// Mitsubishi GX Works2 project: PLC_GROUP_03   PLC: FX3G

// global labels: Global1
VAR_GLOBAL
  petelOriginal AT D1160 : REAL;
  petelCurrent AT D1100 : REAL;
  lemonOriginal AT D1165 : REAL;
  lemonCurrent AT D1105 : REAL;
  meyatzevOriginal AT D1170 : REAL;
  meyatzevCurrent AT D1110 : REAL;
  dubonimOriginal AT D1175 : REAL;
  dubonimCurrent AT D1115 : REAL;
  light7 AT Y007 : BOOL;
  invalidSample AT M4 : BOOL;
  switch5 AT X005 : BOOL;
  no_mlay AT M0 : BOOL;
  switch7 AT X007 : BOOL;
  start_cycle AT X001 : BOOL;
  start_making AT M20 : BOOL;
  TS_0 AT TS0 : BOOL;
  TC_0 AT TC0 : BOOL;
END_VAR
VAR_GLOBAL CONSTANT
  const_50 : INT := 50;
END_VAR
VAR_GLOBAL
  light0 AT Y000 : BOOL;
  sampling AT D1180 : REAL;
  analog_input AT D8280 : INT;
END_VAR
VAR_GLOBAL CONSTANT
  const_400 : REAL := 400.0;
END_VAR
VAR_GLOBAL
  regular_pack AT M1 : BOOL;
  pinuk_pack AT M2 : BOOL;
  mlay_petel_nidrash AT D1120 : REAL;
  mlay_lemon_nidrash AT D1125 : REAL;
  mlay_meyatzev_nidrash AT D1130 : REAL;
  mlay_dubonim_nidrash AT D1135 : REAL;
  no_mlay_petel AT M10 : BOOL;
  no_mlay_lemon AT M11 : BOOL;
  no_mlay_meyatzev AT M12 : BOOL;
  no_mlay_dubonim AT M13 : BOOL;
  switch2 AT X002 : BOOL;
  cooling AT M22 : BOOL;
  light2 AT Y002 : BOOL;
  TC_1 AT TC1 : BOOL;
  TS_1 AT TS1 : BOOL;
  temp_sensor AT X003 : BOOL;
  cool_petel AT D1140 : REAL;
  cool_lemon AT D1145 : REAL;
  mixing AT M24 : BOOL;
  mix_container AT D1150 : REAL;
  mix_time AT D1210 : REAL;
  TC_4 AT TC4 : BOOL;
  TS_4 AT TS4 : BOOL;
  flashing_indicator AT M30 : BOOL;
  TC_2 AT TC2 : BOOL;
  TS_2 AT TS2 : BOOL;
  flash_1 AT Y005 : BOOL;
  flash_2 AT Y006 : BOOL;
  TC_3 AT TC3 : BOOL;
  TS_3 AT TS3 : BOOL;
  finish_mixing AT M40 : BOOL;
  end_work_day AT M5 : BOOL;
  analog_output AT D8282 : INT;
  stock AT D1155 : REAL;
  stock_num AT D1155 : REAL;
END_VAR

// task Task_01 (event TRUE, interval 0, priority 31): POU_01

PROGRAM POU_01
(* structured ladder/FBD written out as ST: instructions are called as NAME(EN, inputs, outputs); _pN, _eN, _tN stand for wires *)
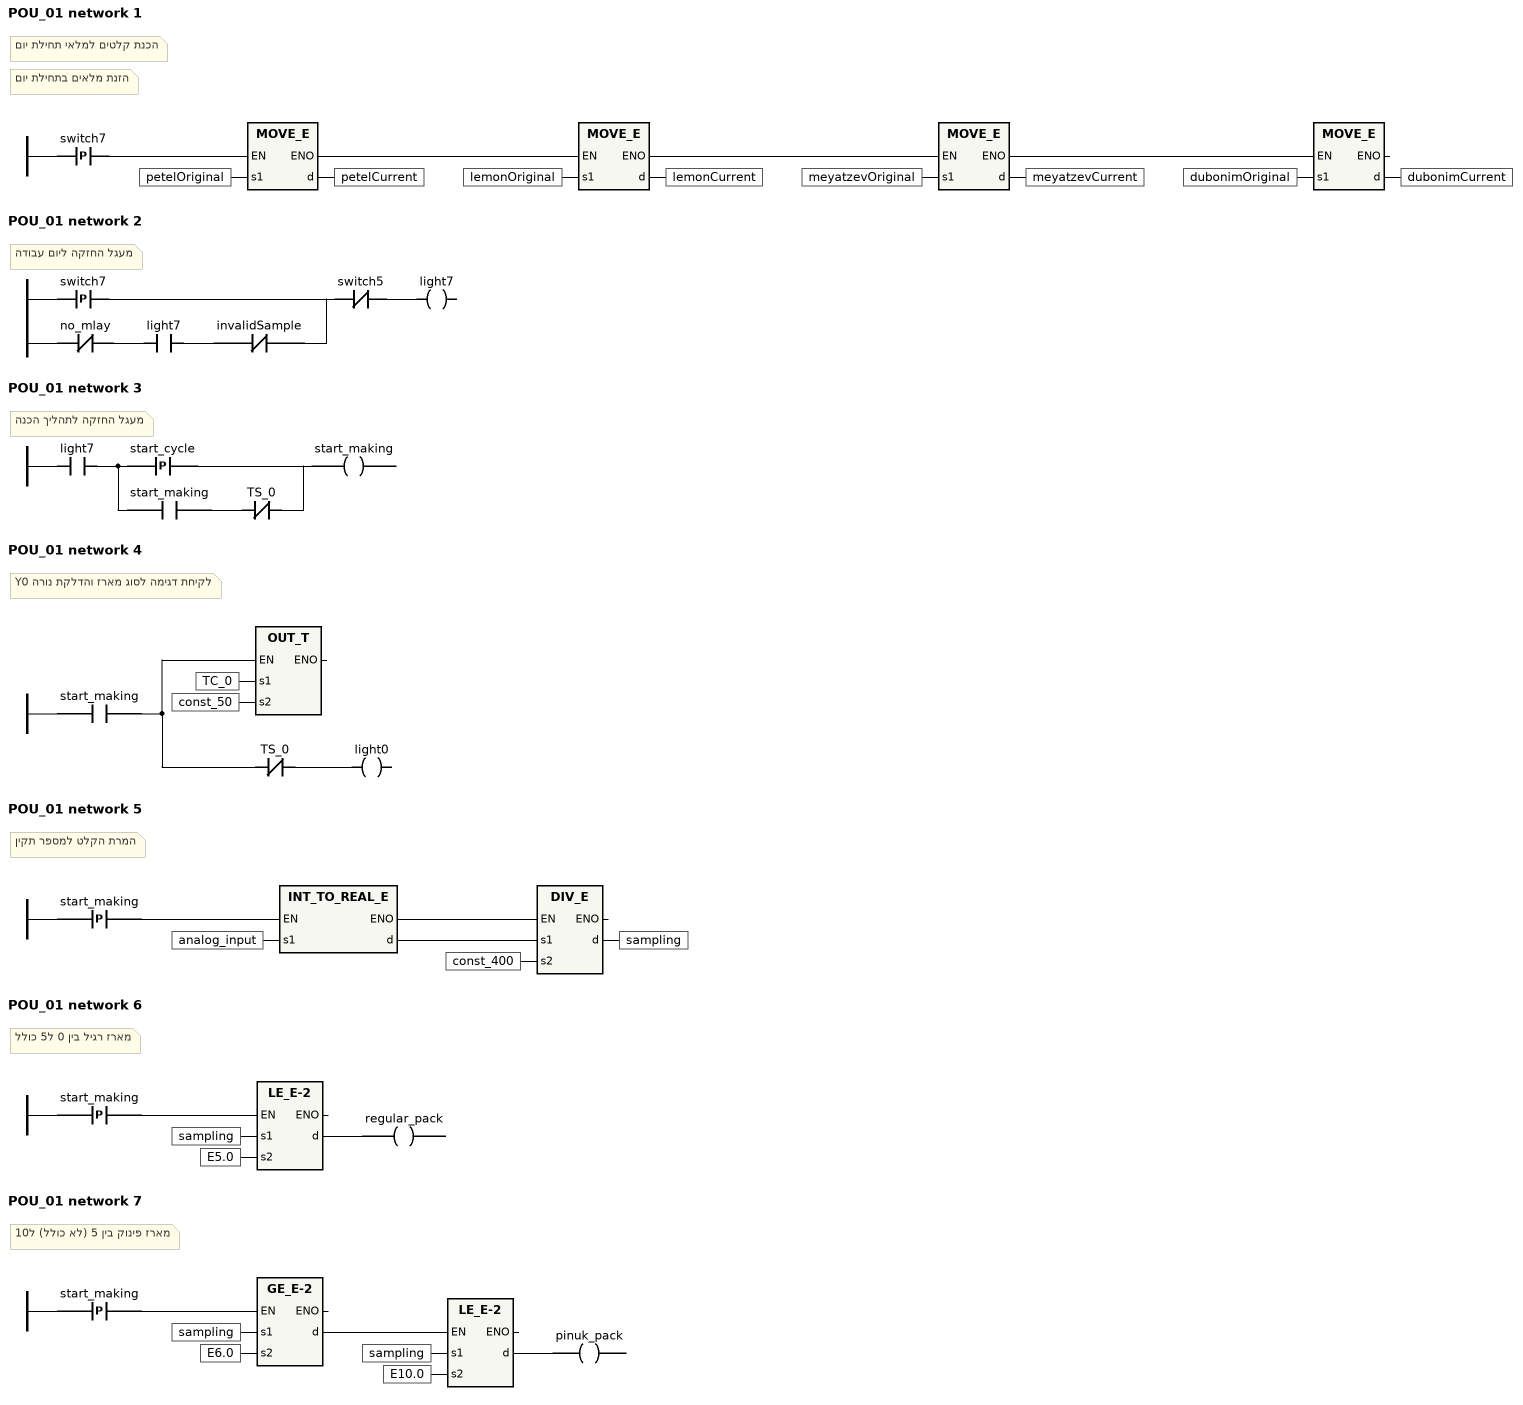
(* network 1 *)
(* הכנת קלטים למלאי תחילת יום *)
(* הזנת מלאים בתחילת יום *)
_e1 := MOVE_E(LDP(TRUE, switch7), petelOriginal, petelCurrent);
_e2 := MOVE_E(_e1, lemonOriginal, lemonCurrent);
_e3 := MOVE_E(_e2, meyatzevOriginal, meyatzevCurrent);
MOVE_E(_e3, dubonimOriginal, dubonimCurrent);
(* network 2 *)
(* מעגל החזקה ליום עבודה *)
light7 := (LDP(TRUE, switch7) OR (NOT no_mlay AND light7 AND NOT invalidSample)) AND NOT switch5;
(* network 3 *)
(* מעגל החזקה לתהליך הכנה *)
start_making := (light7 AND LDP(TRUE, start_cycle)) OR (light7 AND start_making AND NOT TS_0);
(* network 4 *)
(* לקיחת דגימה לסוג מארז והדלקת נורה Y0 *)
OUT_T(start_making, TC_0, const_50);
light0 := start_making AND NOT TS_0;
(* network 5 *)
(* המרת הקלט למספר תקין *)
_e2 := INT_TO_REAL_E(LDP(TRUE, start_making), analog_input, _t1);
DIV_E(_e2, _t1, const_400, sampling);
(* network 6 *)
(* מארז רגיל בין 0 ל5 כולל *)
LE_E(LDP(TRUE, start_making), sampling, E5.0, _t1);
regular_pack := _t1;
(* network 7 *)
(* מארז פינוק בין 5 (לא כולל) ל10 *)
GE_E(LDP(TRUE, start_making), sampling, E6.0, _t1);
LE_E(_t1, sampling, E10.0, _t2);
pinuk_pack := _t2;
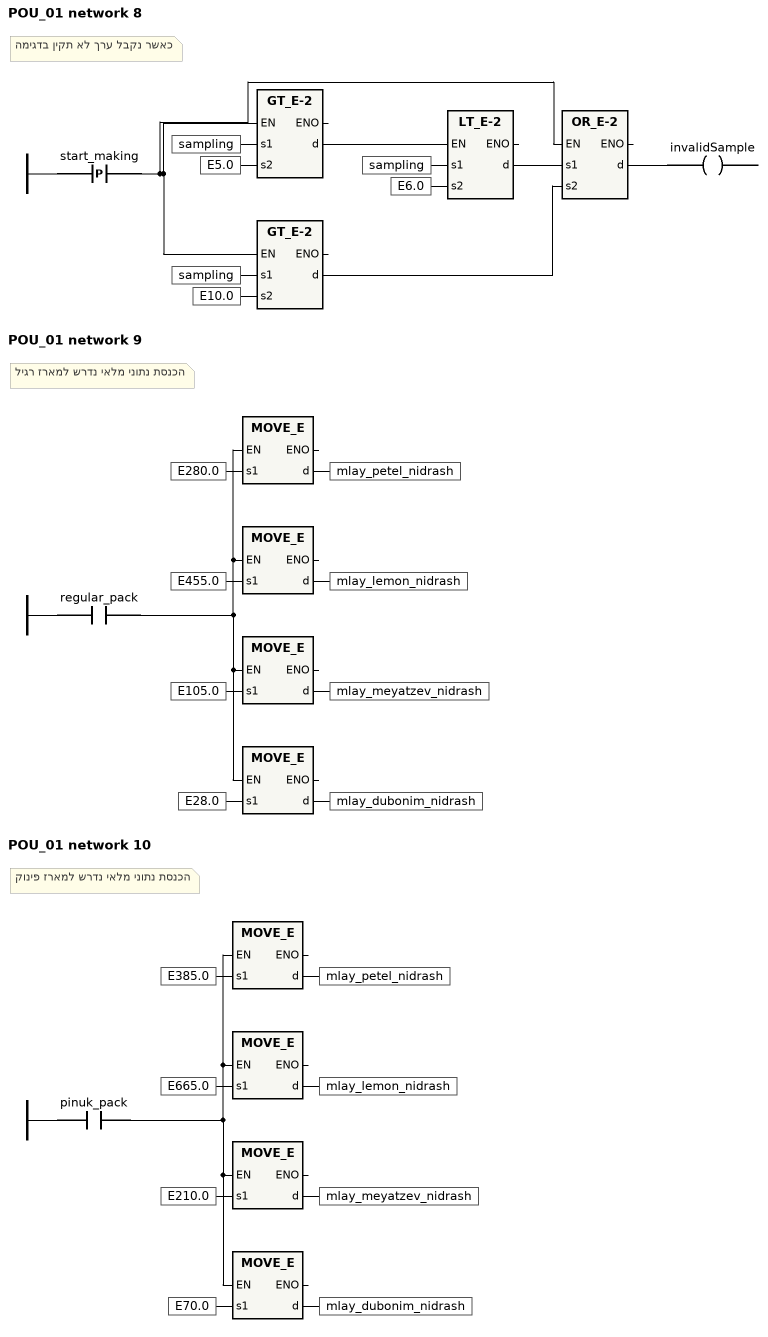
(* network 8 *)
(* כאשר נקבל ערך לא תקין בדגימה *)
_p1 := LDP(TRUE, start_making);
GT_E(_p1, sampling, E5.0, _t2);
LT_E(_t2, sampling, E6.0, _t3);
GT_E(_p1, sampling, E10.0, _t4);
OR_E(_p1, _t3, _t4, _t5);
invalidSample := _t5;
(* network 9 *)
(* הכנסת נתוני מלאי נדרש למארז רגיל *)
MOVE_E(regular_pack, E280.0, mlay_petel_nidrash);
MOVE_E(regular_pack, E455.0, mlay_lemon_nidrash);
MOVE_E(regular_pack, E105.0, mlay_meyatzev_nidrash);
MOVE_E(regular_pack, E28.0, mlay_dubonim_nidrash);
(* network 10 *)
(* הכנסת נתוני מלאי נדרש למארז פינוק *)
MOVE_E(pinuk_pack, E385.0, mlay_petel_nidrash);
MOVE_E(pinuk_pack, E665.0, mlay_lemon_nidrash);
MOVE_E(pinuk_pack, E210.0, mlay_meyatzev_nidrash);
MOVE_E(pinuk_pack, E70.0, mlay_dubonim_nidrash);
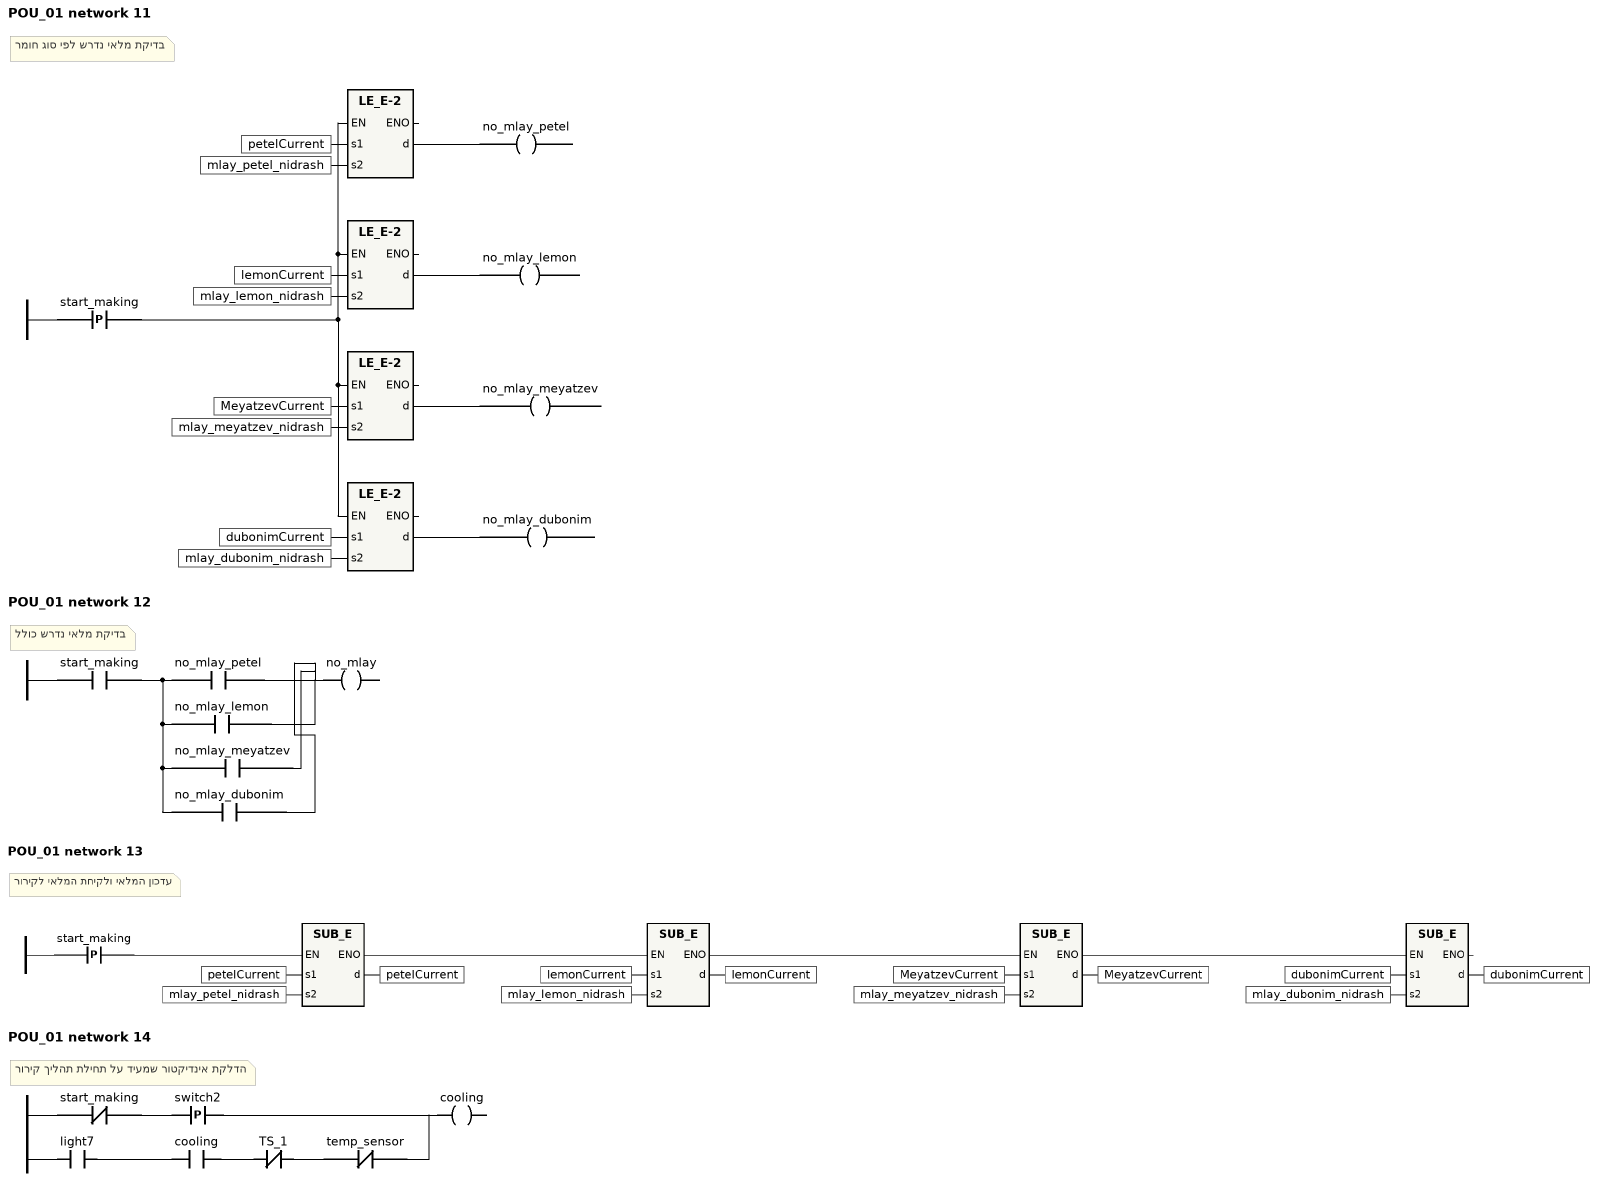
(* network 11 *)
(* בדיקת מלאי נדרש לפי סוג חומר *)
_p1 := LDP(TRUE, start_making);
LE_E(_p1, petelCurrent, mlay_petel_nidrash, _t2);
no_mlay_petel := _t2;
LE_E(_p1, lemonCurrent, mlay_lemon_nidrash, _t3);
no_mlay_lemon := _t3;
LE_E(_p1, MeyatzevCurrent, mlay_meyatzev_nidrash, _t4);
no_mlay_meyatzev := _t4;
LE_E(_p1, dubonimCurrent, mlay_dubonim_nidrash, _t5);
no_mlay_dubonim := _t5;
(* network 12 *)
(* בדיקת מלאי נדרש כולל *)
no_mlay := (start_making AND no_mlay_petel) OR (start_making AND no_mlay_lemon) OR (start_making AND no_mlay_meyatzev) OR (start_making AND no_mlay_dubonim);
(* network 13 *)
(* עדכון המלאי ולקיחת המלאי לקירור *)
_e1 := SUB_E(LDP(TRUE, start_making), petelCurrent, mlay_petel_nidrash, petelCurrent);
_e2 := SUB_E(_e1, lemonCurrent, mlay_lemon_nidrash, lemonCurrent);
_e3 := SUB_E(_e2, MeyatzevCurrent, mlay_meyatzev_nidrash, MeyatzevCurrent);
SUB_E(_e3, dubonimCurrent, mlay_dubonim_nidrash, dubonimCurrent);
(* network 14 *)
(* הדלקת אינדיקטור שמעיד על תחילת תהליך קירור *)
cooling := (NOT start_making AND LDP(TRUE, switch2)) OR (light7 AND cooling AND NOT TS_1 AND NOT temp_sensor);
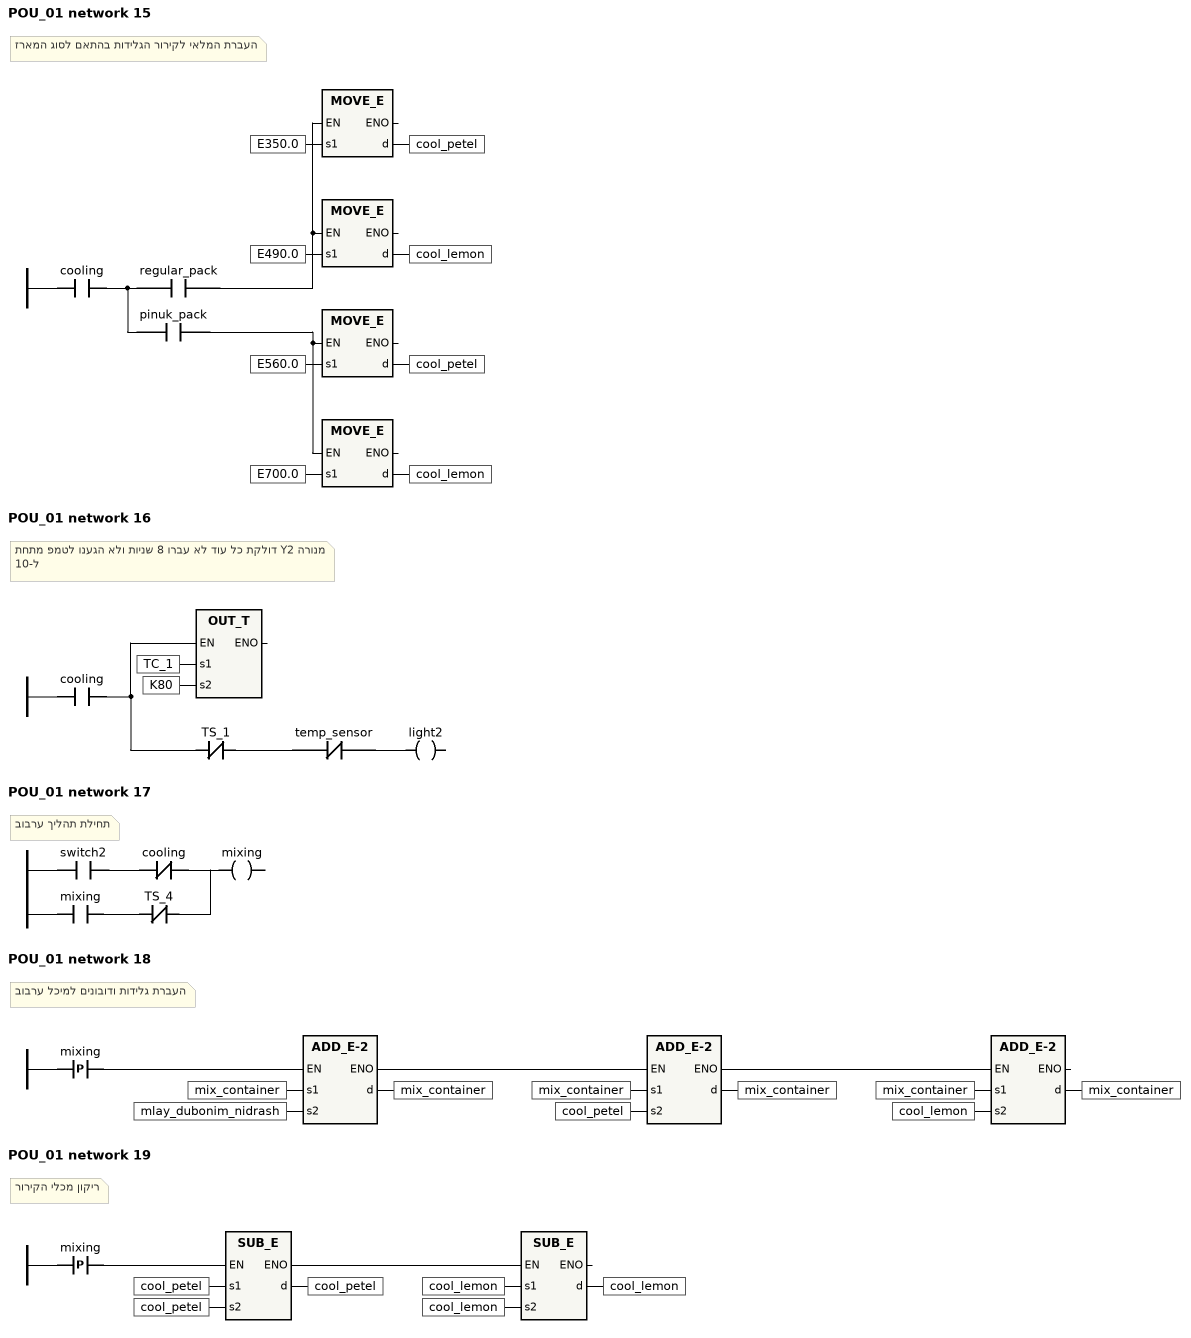
(* network 15 *)
(* העברת המלאי לקירור הגלידות בהתאם לסוג המארז *)
_p1 := cooling AND regular_pack;
MOVE_E(_p1, E350.0, cool_petel);
MOVE_E(_p1, E490.0, cool_lemon);
_p2 := cooling AND pinuk_pack;
MOVE_E(_p2, E560.0, cool_petel);
MOVE_E(_p2, E700.0, cool_lemon);
(* network 16 *)
(* מנורה Y2 דולקת כל עוד לא עברו 8 שניות ולא הגענו לטמפ מתחת ל-10 *)
OUT_T(cooling, TC_1, K80);
light2 := cooling AND NOT TS_1 AND NOT temp_sensor;
(* network 17 *)
(* תחילת תהליך ערבוב *)
mixing := (switch2 AND NOT cooling) OR (mixing AND NOT TS_4);
(* network 18 *)
(* העברת גלידות ודובונים למיכל ערבוב *)
_e1 := ADD_E(LDP(TRUE, mixing), mix_container, mlay_dubonim_nidrash, mix_container);
_e2 := ADD_E(_e1, mix_container, cool_petel, mix_container);
ADD_E(_e2, mix_container, cool_lemon, mix_container);
(* network 19 *)
(* ריקון מכלי הקירור *)
_e1 := SUB_E(LDP(TRUE, mixing), cool_petel, cool_petel, cool_petel);
SUB_E(_e1, cool_lemon, cool_lemon, cool_lemon);
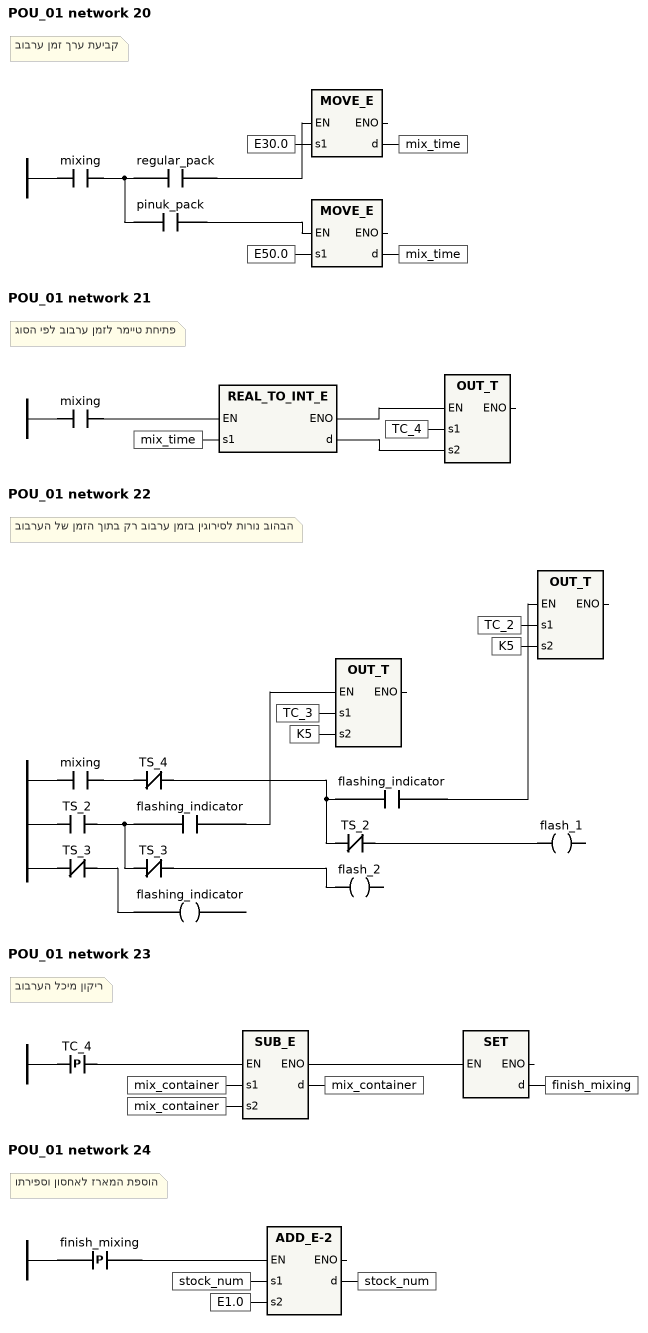
(* network 20 *)
(* קביעת ערך זמן ערבוב *)
MOVE_E(mixing AND regular_pack, E30.0, mix_time);
MOVE_E(mixing AND pinuk_pack, E50.0, mix_time);
(* network 21 *)
(* פתיחת טיימר לזמן ערבוב לפי הסוג *)
_e2 := REAL_TO_INT_E(mixing, mix_time, _t1);
OUT_T(_e2, TC_4, _t1);
(* network 22 *)
(* הבהוב נורות לסירוגין בזמן ערבוב רק בתוך הזמן של הערבוב *)
_p1 := mixing AND NOT TS_4;
OUT_T(_p1 AND flashing_indicator, TC_2, K5);
flash_1 := _p1 AND NOT TS_2;
OUT_T(TS_2 AND flashing_indicator, TC_3, K5);
flash_2 := TS_2 AND NOT TS_3;
flashing_indicator := NOT TS_3;
(* network 23 *)
(* ריקון מיכל הערבוב *)
_e1 := SUB_E(LDP(TRUE, TC_4), mix_container, mix_container, mix_container);
SET(_e1, finish_mixing);
(* network 24 *)
(* הוספת המארז לאחסון וספירתו *)
ADD_E(LDP(TRUE, finish_mixing), stock_num, E1.0, stock_num);
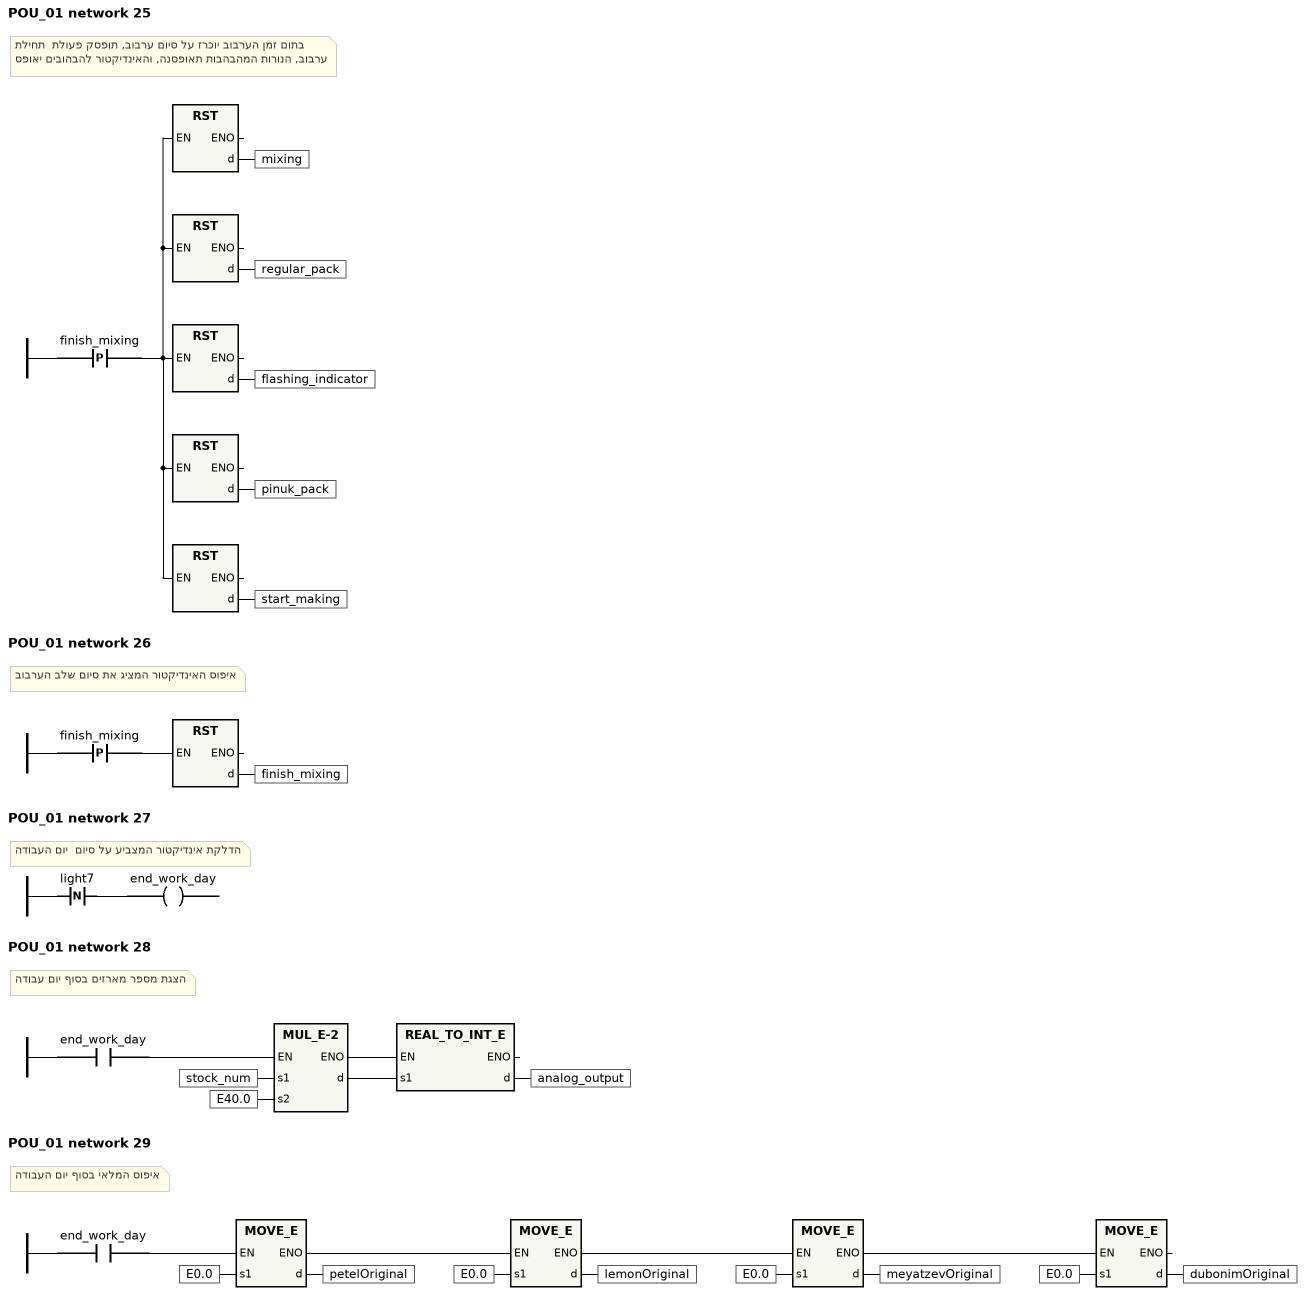
(* network 25 *)
(* בתום זמן הערבוב יוכרז על סיום ערבוב, תופסק פעולת  תחילת ערבוב, הנורות המהבהבות תאופסנה, והאינדיקטור להבהובים יאופס *)
_p1 := LDP(TRUE, finish_mixing);
RST(_p1, mixing);
RST(_p1, regular_pack);
RST(_p1, flashing_indicator);
RST(_p1, pinuk_pack);
RST(_p1, start_making);
(* network 26 *)
(* איפוס האינדיקטור המציג את סיום שלב הערבוב *)
RST(LDP(TRUE, finish_mixing), finish_mixing);
(* network 27 *)
(* הדלקת אינדיקטור המצביע על סיום  יום העבודה *)
end_work_day := LDF(TRUE, light7);
(* network 28 *)
(* הצגת מספר מארזים בסוף יום עבודה *)
_e2 := MUL_E(end_work_day, stock_num, E40.0, _t1);
REAL_TO_INT_E(_e2, _t1, analog_output);
(* network 29 *)
(* איפוס המלאי בסוף יום העבודה *)
_e1 := MOVE_E(end_work_day, E0.0, petelOriginal);
_e2 := MOVE_E(_e1, E0.0, lemonOriginal);
_e3 := MOVE_E(_e2, E0.0, meyatzevOriginal);
MOVE_E(_e3, E0.0, dubonimOriginal);
END_PROGRAM
